FUNCTION TryConvert_SINT_TO_STRING : BOOL
VAR_INPUT
	in : SINT;
	out : REFERENCE TO STRING;
END_VAR

out := SINT_TO_STRING(in);
TryConvert_SINT_TO_STRING := TRUE;

END_FUNCTION

(* stored: Version 1.1.0.1, ProductVersion 3.1.4024.12
   POU TryConvert_SINT_TO_STRING: Id {83caac5b-6c70-47ef-83e6-1e838800c2c3}, SpecialFunc None *)
